FUNCTION_BLOCK FB_Clock
VAR_INPUT
	bEnable : BOOL;
END_VAR
VAR_OUTPUT
	fTime : LREAL;
END_VAR
VAR
	stParameter : ST_Parameters;
END_VAR

IF bEnable THEN
	fTime := fTime + stParameter.fCyclicTime;
ELSE
	fTime := 0.0; 	
END_IF

END_FUNCTION_BLOCK

(* stored: Version 1.1.0.1
   POU FB_Clock: Id {2256c947-436e-4f89-b1da-3b4ee60c3830}, SpecialFunc None *)
